% RSLogix 500 project start_stop_motor.RSS, saved by version 8.30.00.16 %
PROJECT "STASTO"    % processor: Bul.1763 MicroLogix 1100 Series B %

PROGRAM FILES
  LAD 2   4 rungs

DATA FILES
  O0 OUTPUT  4 elements
  I1 INPUT  6 elements
  S2 STATUS  66 elements
  B3 BINARY  1 elements
  T4 TIMER  1 elements
  C5 COUNTER  1 elements
  R6 CONTROL  1 elements
  N7 INTEGER  1 elements
  F8 FLOAT  1 elements

LADDER 2
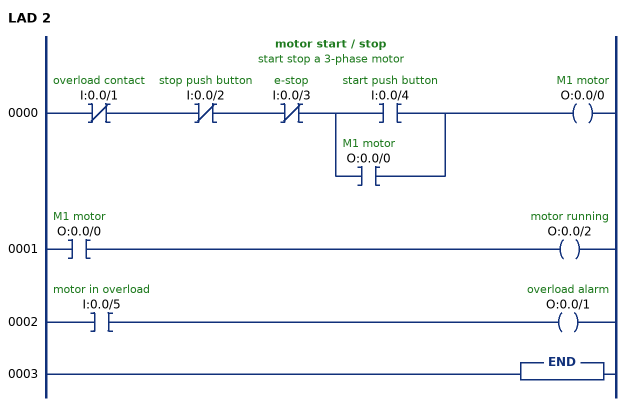
% Rung: 0 %
% TITLE: motor start / stop %
% start stop a 3-phase motor %
SOR XIO I:0.0/1 XIO I:0.0/2 XIO I:0.0/3 BST XIC I:0.0/4 NXB XIC O:0.0/0 BND OTE O:0.0/0 EOR
%   I:0.0/1  "overload contact" %
%   I:0.0/2  "stop push button" %
%   I:0.0/3  "e-stop" %
%   I:0.0/4  "start push button" %
%   O:0.0/0  "M1 motor" %
% Rung: 1 %
SOR XIC O:0.0/0 OTE O:0.0/2 EOR
%   O:0.0/0  "M1 motor" %
%   O:0.0/2  "motor running" %
% Rung: 2 %
SOR XIC I:0.0/5 OTE O:0.0/1 EOR
%   I:0.0/5  "motor in overload" %
%   O:0.0/1  "overload alarm" %
% Rung: 3 %
SOR END EOR
